TYPE "udt_DoorSts"
VERSION : 0.1
// Block: udt_DoorSts
   STRUCT
      OK : Bool;
      NormalStop : Bool;
      SafeStop : Bool;
      EntryEnable : Bool;
      Warning_DoorOpened : Bool;
      Warning_DoorOpenRequest : Bool;
   END_STRUCT;

END_TYPE
